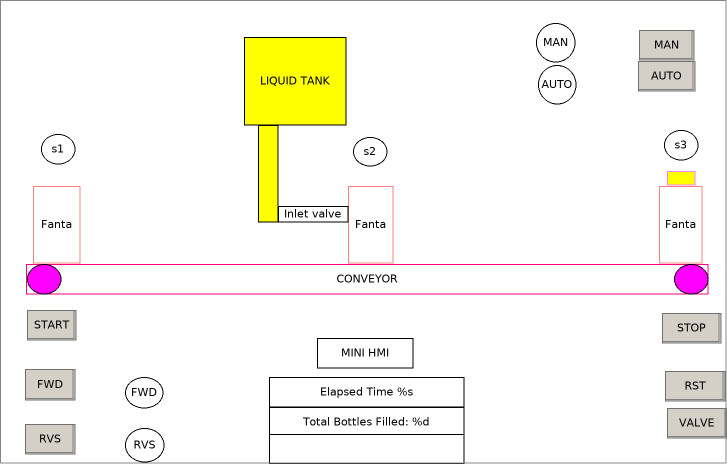
VISUALIZATION FILLER  // 727x464
    Ellipse (41,134 34x30), "s1", colour toggle: MAIN.bSensor1
    Ellipse (353,137 34x29), "s2", colour toggle: MAIN.bSensor2
    Ellipse (664,130 34x30), "s3", colour toggle: MAIN.bSensor3
    RoundedRectangle (33,186 47x77), "Fanta", invisible if: not MAIN.bBottle1
    RoundedRectangle (348,186 45x77), "Fanta", colour toggle: MAIN.bBottle2, invisible if: not MAIN.bBottle2
    RoundedRectangle (659,186 43x77), "Fanta", colour toggle: MAIN.bBottle3, invisible if: not MAIN.bBottle3
    Rectangle (244,37 102x88), "LIQUID TANK"
    Button (662,313 59x30), "STOP"
        OnMouseClick: execute { main.bStopButton:=TRUE; }
    Button (27,310 49x30), "START"
        OnMouseClick: execute { main.bLoadBottle:=true; }
    Button (638,61 57x30), "AUTO"
        OnMouseClick: execute { main.bAutoMode:=TRUE; }
    Button (639,30 55x30), "MAN"
        OnMouseClick: execute { main.bManualMode:=true; }
    Button (665,371 60x30), "RST"
        OnMouseClick: execute { main.bResetButton:=TRUE; }
    Button (667,408 60x30), "VALVE"
        OnMouseClick: execute { main.bInletValve:=TRUE; }
    Button (25,424 50x30), "RVS"
        OnMouseClick: execute { main.bReverseMode:=TRUE; main.bReverseButton:=TRUE; }
    Button (25,369 50x31), "FWD"
        OnMouseClick: execute { main.bForwardMode:=TRUE; main.bForwardButton:=TRUE; }
    Ellipse (536,23 39x39), "MAN", colour toggle: MAIN .bManualLight
    Ellipse (538,65 38x39), "AUTO", colour toggle: MAIN.bAutoLight
    Rectangle (269,377 195x30), "Elapsed Time %s", text variable: MAIN.fbMyTimer.ET
    Rectangle (269,407 195x30), "Total Bottles Filled: %d", text variable: MAIN.iTotalBottles
    Rectangle (269,434 195x30)
    RoundedRectangle (317,338 96x30), "MINI HMI"
    Rectangle (258,125 20x97)
    Rectangle (278,206 70x16), "Inlet valve", colour toggle: MAIN.bInletValve
    RoundedRectangle (26,264 682x30), "CONVEYOR", colour toggle: MAIN.bConveyorMotor
    Ellipse (674,264 34x30)
    Ellipse (27,264 34x30)
    Rectangle (667,171 28x14), invisible if: not MAIN.bBottle3
    Ellipse (125,377 38x31), "FWD", colour toggle: MAIN.bForwardMode
    Ellipse (125,428 39x34), "RVS", colour toggle: MAIN.bReverseMode
END_VISUALIZATION

(* stored: Version 1.1.0.1, ProductVersion 3.1.4024.11
   Visu FILLER: Id {3705eed6-a308-4ddf-a3ca-35f16a36f65d} *)
